// TIA Portal V17 export
// export: Created 2024-10-17T14:16:17.0174027Z, ExportSetting WithDefaults, DisplayName Totally Integrated Automation Portal, DisplayVersion V17 Update 4, DisplayName TIA Portal Openness, DisplayVersion V17 Update 4, DisplayName TIA Portal Version Control Interface, DisplayVersion V17, DisplayName SINAMICS Startdrive Advanced, DisplayVersion V17 Update2, DisplayName SINAMICS Startdrive G130, G150, S120, S150, SINAMICS MV, S210, DisplayVersion V17 Update2, DisplayName SINAMICS Startdrive G110M, G120, G120C, G120D, G120P, G115D, DisplayVersion V17 Update2, DisplayName STEP 7 Professional, DisplayVersion V17 Update 4, DisplayName STEP 7 Safety, DisplayVersion V17, DisplayName WinCC Advanced / Unified PC, DisplayVersion V17 Update 4
TYPE "LPMLV2022_typeAdmin"
TITLE = LPMLV2022_typeAdmin
// Support: tech.team.motioncontrol@siemens.com
// stored: IsFailsafeCompliant false
   STRUCT
      Parameter_REAL { ExternalWritable := 'False'} : Array[0.."LPMLV2022_ADMIN_PARAMETER_REAL_UPPER_LIM"] of "LPMLV2022_typeParameter_REAL";   // Structured Array of Unit/Machine Parameter information for values with REAL data type
      Parameter_STRING { ExternalWritable := 'False'} : Array[0.."LPMLV2022_ADMIN_PARAMETER_STRING_UPPER_LIM"] of "LPMLV2022_typeParameter_STRING";   // Structured Array of Unit/Machine Parameter information for values with STRING data type
      Parameter_LREAL { ExternalWritable := 'False'} : Array[0.."LPMLV2022_ADMIN_PARAMETER_LREAL_UPPER_LIM"] of "LPMLV2022_typeParameter_LREAL";   // Structured Array of Unit/Machine Parameter information for values with LREAL data type
      Parameter_DINT { ExternalWritable := 'False'} : Array[0.."LPMLV2022_ADMIN_PARAMETER_DINT_UPPER_LIM"] of "LPMLV2022_typeParameter_DINT";   // Structured Array of Unit/Machine Parameter information for values with DINT data type
      Parameter_BOOL { ExternalWritable := 'False'} : Array[0.."LPMLV2022_ADMIN_PARAMETER_BOOL_UPPER_LIM"] of "LPMLV2022_typeParameter_BOOL";   // Structured Array of Unit/Machine Parameter information for values with BOOL data type
      Alarm { ExternalWritable := 'False'} : Array[0.."LPMLV2022_ADMIN_ALARM_UPPER_LIM"] of "LPMLV2022_typeEvent";   // Array of Given Size for Machine Alarms. The alarm tags associated to the local interface are typically used as parameters that are displayed or used on the unit locally, for example from an HMI. These alarm parameters can be used to display any alarm, or machine downtime cause that is currently occurring in the system
      AlarmExtent { ExternalWritable := 'False'} : DInt;   // Extent of Alarm Array. The alarm extent is associated with the maximum number of alarms needed for the machine annunciation or reporting
      AlarmHistory { ExternalWritable := 'False'} : Array[0.."LPMLV2022_ADMIN_ALARM_HISTORY_UPPER_LIM"] of "LPMLV2022_typeEvent";   // Array of Given Size for Machine Fault Number and Messaging History. The AlarmHistory array is reserved for alarms that have occurred on the unit/machine and can be sorted in chronological order with the most recently occurring alarmed indexed as Admin.AlarmHistory[0]
      AlarmHistoryExtent { ExternalWritable := 'False'} : DInt;   // Extent of Alarm History Array. The alarm history extent is associated with the maximum number of alarms needed to be archived or tagged as alarm history for the machine
      StopReason { ExternalWritable := 'False'} : "LPMLV2022_typeEvent";   // Machine Stop Reason is typically used for "First Out Fault" Reporting and Other Stoppage Events. The stop reason is the first event captured during an abort, held, suspended or stop event
      Warning { ExternalWritable := 'False'} : Array[0.."LPMLV2022_ADMIN_WARNING_UPPER_LIM"] of "LPMLV2022_typeEvent";   // Machine warnings are for general events that do not cause the machine to stop, but may require operator action as a stoppage may be imminent. Warnings are not typically stored in history
      WarningExtent { ExternalWritable := 'False'} : DInt;   // Extent of Warning Array. The warning extent is associated with the maximum number of warnings needed to be archived or tagged as warnings for the machine
      ModeTimeCurrent { ExternalWritable := 'False'} : DInt;   // Current Mode Time. This tag represents the current amount of time (in seconds) spent in the current Mode as indicated by Status.UnitModeCurrent. The value will start from 0 every time the Mode is changed
      StateTimeCurrent { ExternalWritable := 'False'} : DInt;   // Current State Time. This tag represents the current amount of time (in seconds) spent in the current State as indicated by Status.StateCurrent. The value will start from 0 every time the State is changed
      CumulativeTimes { ExternalWritable := 'False'} : Array[0.."LPMLV2022_ADMIN_CUMULATIVE_TIMES_UPPER_LIM"] of "LPMLV2022_typeCumulativeTimes";   // Structured Array of Timer Values. This tag represents a collection of accumulated time (in seconds) spent in any defined state of any defined mode
      ProductData { ExternalWritable := 'False'} : Array[0.."LPMLV2022_ADMIN_PRODUCT_DATA_UPPER_LIM"] of "LPMLV2022_typeProductData";   // Structured array of Product Stream Data. This tag represents a collection of information about each unique input or output product stream of the machine unit. The extent of the array is typically limited to the maximum number of input and output product streams
      MachDesignSpeed { ExternalWritable := 'False'} : Real;   // Machine Design Speed. This tag represents the maximum design speed of the machine in primary packages per minute for the package configuration being run. This speed is NOT the maximum speed as specified by the manufacturer, but rather the speed of the machine is designed to run in its installed environment
      DisabledStatesCfg { ExternalWritable := 'False'} : Array[0.."LPMLV2022_ADMIN_NUMBER_OF_MODES_UPPER_LIM"] of DWord;   // An array reflecting the Disabled States Configuration for all defined Modes. The array index represents the Mode number. Bit locations within the DWORD value represent State numbers. A value of 1 in a bit location indicates that the corresponding state number is disabled. State 0 is an Undefined State, therefore bit 0 is unused
      CurDisabledStates { ExternalWritable := 'False'} : DWord;   // Reflects the disabled states for the current Mode (Status.UnitModeCurrent). State numbers are represented by bit location. A value of 1 in a certain bit location indicates that the corresponding state number is disabled. State 0 is an Undefined State, therefore bit 0 is unused
      EnabledModesCfg { ExternalWritable := 'False'} : DWord;   // An element reflecting the Enabled Modes Configuration for the unit/machine. Bit locations within the DWORD represent Mode numbers. A value of 1 in a bit location [0-31] indicates that the corresponding Mode number is enabled. Mode 0 is an Invalid Mode, therefore bit 0 is unused
      ModeTransitionCfg { ExternalWritable := 'False'} : Array[0.."LPMLV2022_ADMIN_NUMBER_OF_MODES_UPPER_LIM"] of DWord;   // An array reflecting the Mode Transition Configuration for all modes of the unit/machine. The array index represents the Mode number. Bit locations within the DWORD value represent State numbers. A value of 1 in a bit location indicates that a mode transition from the corresponding state number is allowed
      PLCDateTime { ExternalWritable := 'False'} : "LPMLV2022_typeDateTime";   // Current Date and Time of the Programmable Logic Controller
      PLCDateTimeDTL { ExternalWritable := 'False'} : DTL;   // Current Date and Time (DTL) of the Programmable Logic Controller
   END_STRUCT;
END_TYPE
